(* CODESYS project Lamp_student.project

Project tree, tasks and I/O mapping:
  Device : CODESYS Control Win V3, 3S - Smart Software Solutions GmbH, version 3.5.17.10
    application Application
      libraries: Standard, * (System)
      task MainTask (cyclic, interval 100 ms, priority 1) calls PLC_PRG
      program PLC_PRG [ST]
      visualisation Visualization
      image pool ImagePool
  text list GlobalTextList
  5ce3da45-db07-42e7-a21c-a00fff4ed8f6|E:\ONO.png
  5ce3da45-db07-42e7-a21c-a00fff4ed8f6|E:\OFF3.png
*)

// Device/Application/PLC_PRG
PROGRAM PLC_PRG
VAR_INPUT
	Button :BOOL;
END_VAR

VAR_OUTPUT
	Lamp :BOOL;
END_VAR

IF (Button = 1) THEN
	Lamp := 1; // Jos Input (Button) on 1 niin Asetetaan Lampun arvoksi TRUE eli 1.
ELSE
	LAMP := 0; // Jos Input (Button) on 0 (Tai mikä vaan muu. Voitaisiin myös laittaa ELSEIF (Button = 0) niin Asetetaan Lampun arvoksi FALSEE eli 0.
END_IF;

END_PROGRAM

// Device/Application/Visualization
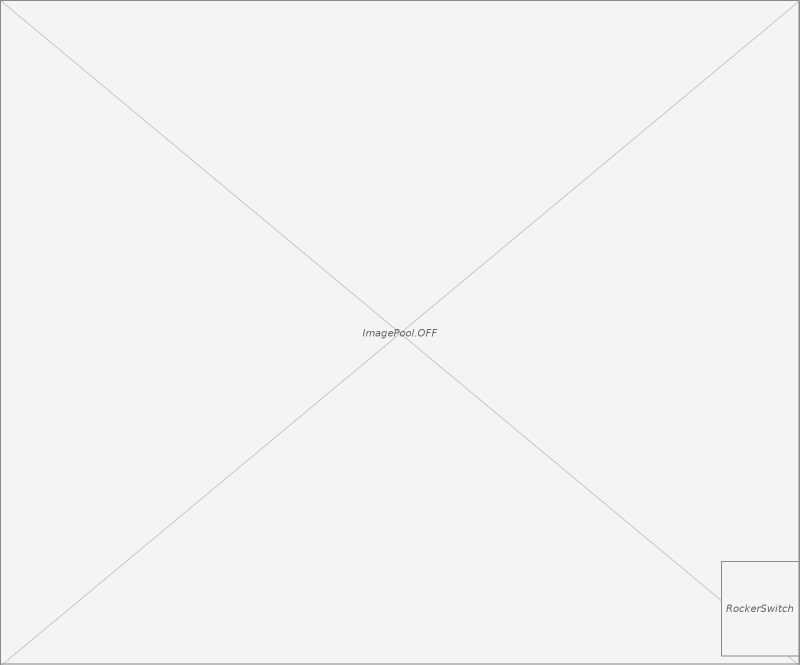
VISUALIZATION Visualization  // 800x665
    Image (0,0 800x666), image: ImagePool.ON
    Image (0,0 800x666), invisible if: PLC_PRG.Lamp, image: ImagePool.OFF
    RockerSwitch (721,561 78x95), variable: PLC_PRG.Button, behaviour: TOGGLE, style: Switch-RockerSwitch-Gray
END_VISUALIZATION
